SUBAPPLICATION Uebung_219_AULI (* Standard IEC 61131-3 AULI_FB_CTD (Adapter Version, Rückwärtszähler, ULINT) mit Terminal-Ausgabe *)
  (* Standard: 61131-3; Description: Copyright (c) 2026 Meisterschulen am Ostbahnhof This program and the accompanying materials are made available under the terms of the Eclipse Public License 2.0 which is available at https://www.eclipse.org/legal/epl-2.0/ SPDX-License-Identifier: EPL-2.0 *)
  (* Version 1.2, 2026-05-13, Franz Höpfinger, Meisterschulen am Ostbahnhof, Added AULI_ULINT_TO_ULI init block connected to PV *)
  (* Version 1.1, 2026-04-21, Franz Höpfinger, Meisterschulen am Ostbahnhof, Added terminal output for counter value *)
  (* Version 1.0, 2026-04-21, Franz Höpfinger, Meisterschulen am Ostbahnhof, initial API and implementation (Adapter version) *)
  PACKAGE Uebungen;
  IMPORT Uebungen::const::UT::DefaultPool::OutputNumber_N1;
  IMPORT logiBUS::io::DI::logiBUS_DI::Input_I1;
  IMPORT logiBUS::io::DI::logiBUS_DI::Input_I2;
  IMPORT logiBUS::io::DQ::logiBUS_DO::Output_Q1;
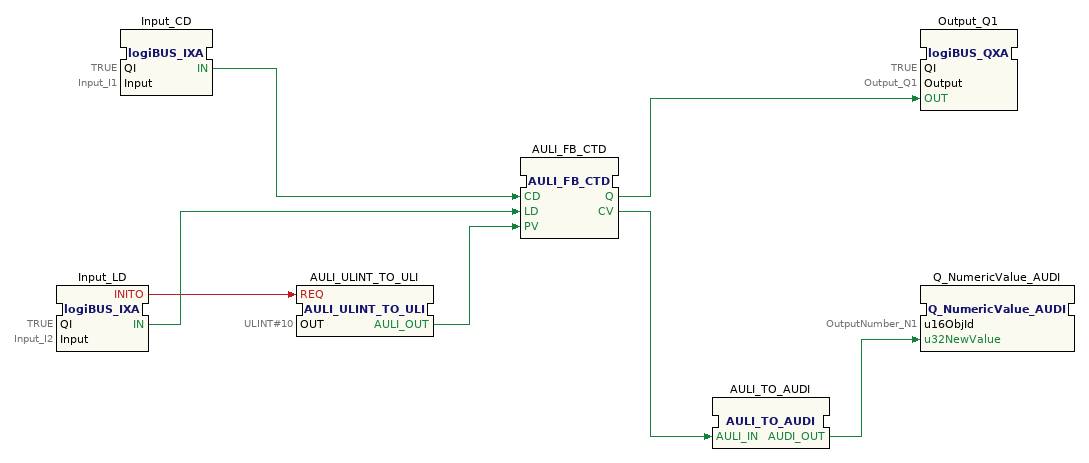
  FBS
    AULI_FB_CTD : adapter::iec61131::counters::AULI_FB_CTD;
    AULI_ULINT_TO_ULI : adapter::conversion::unidirectional::AULI_ULINT_TO_ULI(OUT := ULINT#10);
    Input_CD : logiBUS::io::DI::logiBUS_IXA(QI := TRUE, Input := Input_I1);
    Input_LD : logiBUS::io::DI::logiBUS_IXA(QI := TRUE, Input := Input_I2);
    Output_Q1 : logiBUS::io::DQ::logiBUS_QXA(QI := TRUE, Output := Output_Q1);
    AULI_TO_AUDI : adapter::conversion::unidirectional::AULI_TO_AUDI;
    Q_NumericValue_AUDI : isobus::UT::Q::Q_NumericValue_AUDI(u16ObjId := OutputNumber_N1);
  END_FBS
  EVENT_CONNECTIONS
    Input_LD.INITO TO AULI_ULINT_TO_ULI.REQ;
  END_CONNECTIONS
  ADAPTER_CONNECTIONS
    Input_CD.IN TO AULI_FB_CTD.CD;
    Input_LD.IN TO AULI_FB_CTD.LD;
    AULI_FB_CTD.Q TO Output_Q1.OUT;
    AULI_FB_CTD.CV TO AULI_TO_AUDI.AULI_IN;
    AULI_TO_AUDI.AUDI_OUT TO Q_NumericValue_AUDI.u32NewValue;
    AULI_ULINT_TO_ULI.AULI_OUT TO AULI_FB_CTD.PV;
  END_CONNECTIONS
END_SUBAPPLICATION
